(* CODESYS project Motor.project
   Title: Motor
   Version: 0.0.0.0
   Author: Enes

Project tree, tasks and I/O mapping:
  MyController : TM241C24T/U, Schneider Electric, order no. TM241C24T/U, version 4.0.6.18
    application Application
      task MAST (cyclic, interval 20 ms, priority 15, watchdog 100 ms x 1) calls POU
      global variables GVL
      program POU [LD]
    DI : Digital Inputs, Schneider Electric, version 4.0.6.18
        settings: IOs Usage = 1
        input  iwDI_IW0 : WORD  // IW0
        input  ibDI_IB1 : BYTE  // IB1
    DQ : Digital Outputs, Schneider Electric, version 4.0.6.18
        settings: Outputs Usage = 3
        output qwDQ_QW0 : WORD  // QW0
        output qbDQ_QB1 : BYTE  // QB1
    Counters : Counters, Schneider Electric, version 4.0.6.18
    Pulse_Generators : Pulse Generators, Schneider Electric, version 4.0.6.18
        settings: Instance name = 'PTO_0'; PROBE input History = 'old=1 new=-1'; INDEX input History = 'old=0 new=-1'; REF input History = 'old=-1 new=0'; B output History = 'old=-1 new=1'; A output History = 'old=-1 new=0'; Temporary Instance name = 'PTO_0'
    Cartridge_1 : Cartridge, Schneider Electric, version 4.0.6.18
    IO_Bus : IO bus - TM3, Schneider Electric, version 4.0.6.18
    COM_Bus : COM bus, Schneider Electric, version 4.0.6.18
    Serial_Line_1 : Serial line, Schneider Electric, version 4.0.6.18
      SoMachine_Network_Manager : SoMachine-Network Manager, Schneider Electric, version 4.0.0.2
    Serial_Line_2 : Serial line, Schneider Electric, version 4.0.6.18
      Modbus_Manager : Modbus Manager, Schneider Electric, version 4.0.0.2
*)

// MyController/Application/GVL
VAR_GLOBAL
END_VAR

// MyController/Application/POU
PROGRAM POU
VAR
	MC_Power: MC_Power_PTO;
	Start: BOOL;
	MC_Reset: MC_Reset_PTO;
	Reset_En: BOOL;
	MC_Home: MC_Home_PTO;
	Home: BOOL;
	Dir: MC_DIRECTION;
	Pos: DINT;
	Mode: PTO_HOMING_MODE;
	H_Speed: DINT;
	L_Speed: DINT;
	Acc: DINT;
	Dec: DINT;
	Offset: DINT;
	MC_MoveVelocity: MC_MoveVelocity_PTO;
	Vel_En: BOOL;
	MC_Stop: MC_Stop_PTO;
	Motion_Stop: BOOL;
END_VAR

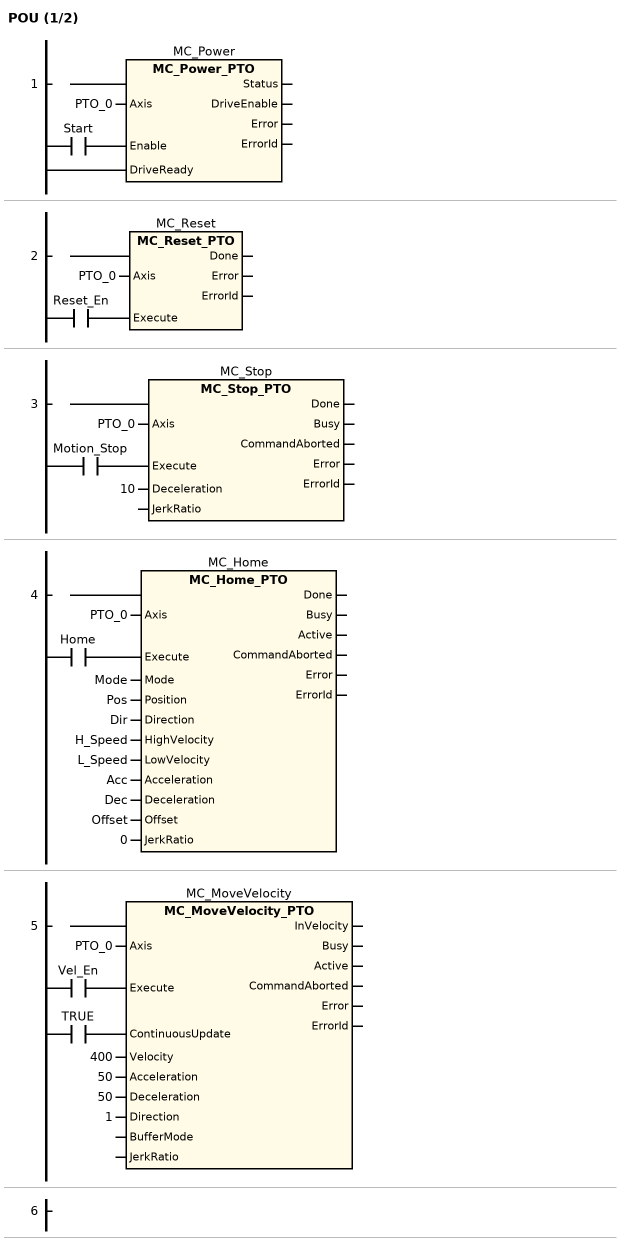
// NETWORK 1
MC_Power(Axis := PTO_0, Enable := Start, DriveReady := TRUE); // MC_Power_PTO

// NETWORK 2
MC_Reset(Axis := PTO_0, Execute := Reset_En); // MC_Reset_PTO

// NETWORK 3
MC_Stop(Axis := PTO_0, Execute := Motion_Stop, Deceleration := 10); // MC_Stop_PTO

// NETWORK 4
MC_Home(
    Axis := PTO_0,
    Execute := Home,
    Mode := Mode,
    Position := Pos,
    Direction := Dir,
    HighVelocity := H_Speed,
    LowVelocity := L_Speed,
    Acceleration := Acc,
    Deceleration := Dec,
    Offset := Offset,
    JerkRatio := 0); // MC_Home_PTO

// NETWORK 5
MC_MoveVelocity(
    Axis := PTO_0,
    Execute := Vel_En,
    ContinuousUpdate := TRUE,
    Velocity := 400,
    Acceleration := 50,
    Deceleration := 50,
    Direction := 1); // MC_MoveVelocity_PTO

// NETWORK 6

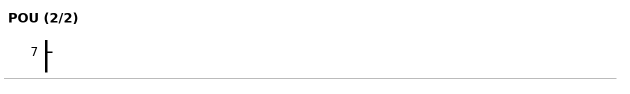
// NETWORK 7

END_PROGRAM
